// TIA Portal V20 export
VAR_GLOBAL   // PLC tag table "LGR_Const_Equip_Mode"
END_VAR
VAR_GLOBAL CONSTANT   // user constants
   MODE_BOOT : Word := 16#0000;
   MODE_INIT : Word := 16#0001;   // X0
   MODE_MAINT : Word := 16#0002;   // X1
   MODE_STANDBY : Word := 16#0004;   // X2
   MODE_MANUAL : Word := 16#0008;   // X3
   MODE_READY : Word := 16#0010;   // X4
   MODE_AUTO : Word := 16#0020;   // X5
   MODE_RESERVED : Word := 16#0040;   // X6
   MODE_FAULT : Word := 16#0080;   // X7
   MODE_TEACH : Word := 16#0100;
END_VAR
